GLOBALCONSTANTS NVS_Keys (* Global constants *)
  (* Standard: 61499-1 *)
  (* Version 1.0, 2024-02-25, franz *)
  VAR_GLOBAL CONSTANT
    Key_Pflanzabstand_Store : STRING := 'K_I1';
    Key_Luftversatz_Store : STRING := 'K_I2';
    Key_Wasserversatz_Store : STRING := 'K_I3';
    Key_Granulatversatz_Store : STRING := 'K_I4';
    Key_Arbeitsminuten_Store : STRING := 'K_I5';
    Key_Einsatzdauer_Stunden_Store : STRING := 'K_I6';
    Key_Einsatzdauer_Minuten_Store : STRING := 'K_I7';
    Key_Baumzaehler_Store : STRING := 'Baumzaehler';
    Key_Summer_Dauer_Store : STRING := 'K_I14';
    Key_Granulat_Dauer_Store : STRING := 'K_I15';
    Key_Luft_Dauer_Store : STRING := 'K_I16';
    Key_Wasser_Dauer_Store : STRING := 'K_I_17';
    Key_VDS_Store : STRING := 'K_I_18';
    Key_WBSD_Store : STRING := 'K_I_19';
    Key_GBSD_Store : STRING := 'K_I_20';
    Key_MSS_Store : STRING := 'K_I_21';
    Key_NMEA_Store : STRING := 'K_I_22';
    Key_Summer_Reset_Store : STRING := 'K_I_23';
  END_VAR
END_GLOBALCONSTANTS
